FUNCTION_BLOCK EL6614
VAR
	{attribute addProperty Name "Info data"}
	_infoData : InfoDataAds;
END_VAR

END_FUNCTION_BLOCK

(* stored: Version 1.1.0.1, ProductVersion 3.1.4024.9
   POU EL6614: Id {311c3909-3d81-0f08-206f-35a5e07b9f03}, SpecialFunc None *)
